ABB RobotStudio station: Pick_Place_Simulation.rsstnx

Station Pick_Place_Simulation (saved by RobotStudio 25.2.11266.1)
Controller IRB120_3_58
  mechanical unit ROB_1: IRB120_3_58__01, 6 joints, base frame (0, 0, 0) mm
Layout (positions relative to the parent item):
  - IRB120_3_58__01 [mechanism, from %ABB.RobotStudio.Models.IRB120%\IRB120_3_58_G_01.rslib] at (0, 0, 0) mm; joint values [0.3969, 0.1483, 0.6552, 0, 0.7633, 0] (rad or m)
  - Smart_Gripper_Servo_Fingers [mechanism, from %ABB.RobotStudio.Models.SmartGripper%\ABB_Smart_Gripper_Servo_Fingers.rslib] at (276.89, 116.04, 316.25) mm, rotated rx 180 ry 0.23 rz -157.26 deg; joint values [0.0045] (rad or m)
  - LineSensor [smart component, from Components\LineSensor.rslib] at (277.31, 116.22, 202.05) mm, rotated rx 180 ry 0.23 rz -157.26 deg
      properties: Start=[0 0 0]; End=[0 0 0.025]; Length=0.025; Radius=0.00425531914893617; Tag=(none); SenseMultiple=false; SensedPart=peg; SensedPoint=[0.171299957275391 0.00349145174026489 0.240397979736328]
    - _sensorPart_ [part], size 8.5 x 8.5 x 25 mm
  - Attacher [smart component, from Components\Attacher.rslib]
      properties: Parent=IRB120_3_58__01; Flange=0; Child=peg; Mount=false; Offset=[0 0 0]; Orientation=[0 0 0]
  - Detacher [smart component, from Components\Detacher.rslib]
      properties: Child=peg; KeepPosition=true
  - PoseMover [smart component, from Components\PoseMover.rslib]
      properties: Mechanism=Smart_Gripper_Servo_Fingers; Pose=2; Duration=0
  - PoseMover_2 [smart component, from Components\PoseMover.rslib]
      properties: Mechanism=Smart_Gripper_Servo_Fingers; Pose=3; Duration=0
  - Plate_A [part] at (232.94, 71.16, 150) mm, size 150 x 150 x 20 mm
  - Plate_B [part] at (198.28, -131.52, 150) mm, rotated rx 0 ry 0 rz -30.88 deg, size 150 x 150 x 20 mm
  - peg [part] at (277.81, 116.04, 165.61) mm, size 9.7 x 9.7 x 20 mm
Attachment: Smart_Gripper_Servo_Fingers is attached to IRB120_3_58__01 / Link6
Attachment: LineSensor is attached to Smart_Gripper_Servo_Fingers / HandBase
Attachment: peg is attached to IRB120_3_58__01 / Link6
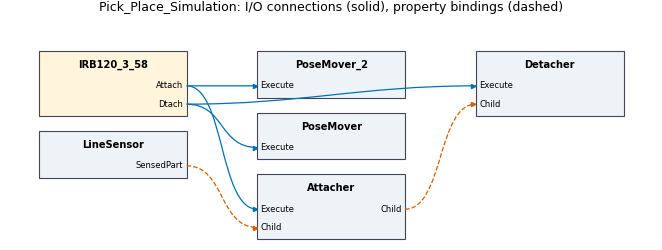
Station logic (signal -> signal, property => property):
  IRB120_3_58.Attach -> Attacher.Execute
  IRB120_3_58.Dtach -> Detacher.Execute
  IRB120_3_58.Attach -> PoseMover_2.Execute
  IRB120_3_58.Dtach -> PoseMover.Execute
  LineSensor.SensedPart => Attacher.Child
  Attacher.Child => Detacher.Child
Targets, tools, work objects and paths stored in the station, written as RAPID:
! task T_ROB1
MODULE CalibData
  PERS tooldata Servo:=[TRUE,[[0,0,114.2],[1,0,0,0]],[0.215,[8.7,12.3,49.2],[1,0,0,0],0.00021,0.00024,0.00009]];
  TASK PERS wobjdata pegA_wb:=[FALSE,TRUE,"",[[232.95217528,71.351942285,170],[0.999999321,-0.000950744,-0.000000641,0.000673854]],[[0,0,0],[1,0,0,0]]];
  TASK PERS wobjdata pegB_wb:=[FALSE,TRUE,"",[[275.064830971,-2.910289774,170.005053754],[0.964289802,0.000030046,0.000109395,-0.264849326]],[[0,0,0],[1,0,0,0]]];
ENDMODULE

! task T_ROB1
MODULE Module1
  CONST num delayTime:=0.5;
  PROC main()
    WaitTime delayTime;
    PulseDO Dtach;
  ENDPROC
ENDMODULE

